PROGRAM MAIN
VAR
END_VAR

END_PROGRAM

(* stored: Version 1.1.0.1
   POU MAIN: Id {35885d34-60cd-4bfd-98da-527d7ce5f47c} *)
